Yaskawa INFORM job: HOME_ROBO_GUN.JBI

/JOB
//NAME HOME_ROBO_GUN
///FOLDERNAME HOME
//POS
///NPOS 0,0,0,1,0,1
///TOOL 0
///POSTYPE PULSE
///PULSE
P00010=140050,-126820,-84504,14231,87660,95695
EX00010=56001
//INST
///DATE 2022/06/13 03:45
///ATTR SC,RW
///GROUP1 RB1,ST1
NOP
EDTLCK MOVJ P010 EX010 VJ=100.00  //HOME
END
